FUNCTION_BLOCK FB_UAreadMock_BoolChangesToTrue IMPLEMENTS I_OPCUA_Read
VAR_INPUT
END_VAR
VAR_OUTPUT
END_VAR
VAR
END_VAR

{warning 'add method implementation '}
METHOD start : BOOL
VAR_INPUT
	Execute	: BOOL;
	ConnectionHdl	: DWORD;
	NodeHdl	: DWORD;
	stNodeAddInfo	: Tc3_PLCopen_OpcUa.ST_UANodeAdditionalInfo;
	pVariable	: PVOID;
	cbData	: UDINT;
	Timeout	: TIME := DEFAULT_ADS_TIMEOUT;
END_VAR
VAR_OUTPUT
	Done	: BOOL;
	Busy	: BOOL;
	Error	: BOOL;
	ErrorID	: UDINT;
	cbData_R	: UDINT;
END_VAR
IF execute THEN
	MEMSET(pVariable,1,SIZEOF(cbData));
	done := TRUE;
END_IF
END_METHOD

END_FUNCTION_BLOCK

(* stored: Version 1.1.0.1, ProductVersion 3.1.4024.9
   POU FB_UAreadMock_BoolChangesToTrue: Id {cbba6015-d072-4f3f-9063-45e2840aa17c}, SpecialFunc None
   Method start: Id {0b163bc4-4f9a-4ca0-a6f6-219381902035} *)
